FUNCTION F_rPressure : WORD
VAR_INPUT
	iRawVoltage : INT;
END_VAR
VAR
END_VAR

(* Transducer voltage to pressure *)
(* Add formula in here *)
F_rPressure := INT_TO_WORD((iRawVoltage*3000)/32767);

END_FUNCTION

(* stored: Version 1.1.0.1, ProductVersion 3.1.0.24
   POU F_rPressure: Id {be680594-3bc8-4d10-9c84-f2a20035e519} *)
